// TIA Portal V19 export
FUNCTION_BLOCK "SAMPLE_BLOCK"   // FB1, LAD
TITLE = Example Function Block - ie, Multiple Motors Start / Stop
{ S7_Optimized_Access := 'TRUE' }
// stored: MemoryReserve 100, SetENOAutomatically false
BEGIN

REGION Network 1: Drive 1 - Latching
   // Motor 1
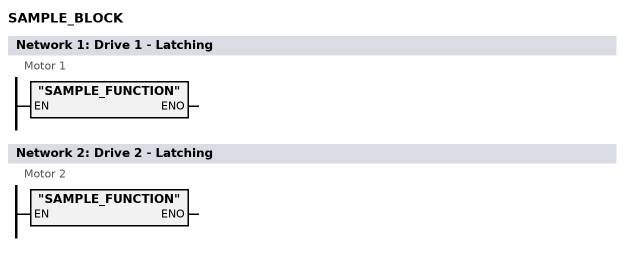
   RUNG wire#powerrail
      "SAMPLE_FUNCTION"()
   END_RUNG
   // the same network as SCL:
   "SAMPLE_FUNCTION"();
END_REGION

REGION Network 2: Drive 2 - Latching
   // Motor 2
   RUNG wire#powerrail
      "SAMPLE_FUNCTION"()
   END_RUNG
   // the same network as SCL:
   "SAMPLE_FUNCTION"();
END_REGION
END_FUNCTION_BLOCK
